{attribute 'qualified_only'}
{attribute 'strict'}
TYPE eTcoOscilatingConveyorStatus :
(
	None:=0,
	Feeding:=1,
	Oscilating:=2,
	ReadyToPick:=3,
	Error:=4

);
END_TYPE

(* stored: Version 1.1.0.1
   DUT eTcoOscilatingConveyorStatus: Id {92e9a479-149e-42d4-86b4-bd589c9656f7} *)
